FUNCTION_BLOCK Resource2
  (* Version 1.0, 2008-11-05, Goran Cengic, Chalmers *)
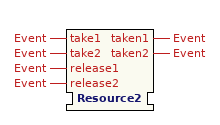
  EVENT_INPUT
    take1;
    take2;
    release1;
    release2;
  END_EVENT
  EVENT_OUTPUT
    taken1;
    taken2;
  END_EVENT
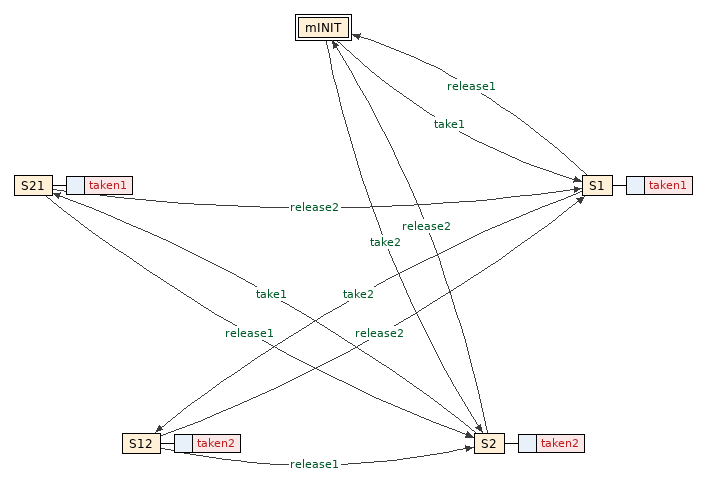
  EC_STATES
    mINIT;
    S1 : -> taken1;
    S2 : -> taken2;
    S12 : -> taken2;
    S21 : -> taken1;
  END_STATES
  EC_TRANSITIONS
    mINIT TO S1 := take1;
    S1 TO mINIT := release1;
    S1 TO S12 := take2;
    S12 TO S1 := release2;
    S12 TO S2 := release1;
    mINIT TO S2 := take2;
    S2 TO mINIT := release2;
    S2 TO S21 := take1;
    S21 TO S2 := release1;
    S21 TO S1 := release2;
  END_TRANSITIONS
END_FUNCTION_BLOCK
